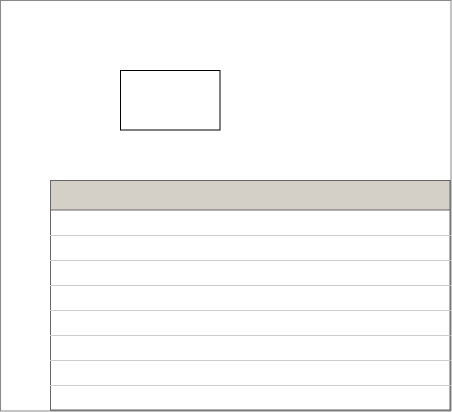
VISUALIZATION test  // 452x412
    Rectangle (120,70 100x60), colour toggle: MAIN.Q
    Table (50,180 400x230), data array: MAIN.arrWaarde
        p2232123230: MAIN.arrWaarde[1, INDEX]
        p511219082: MAIN.arrWaarde[2, INDEX]
END_VISUALIZATION

(* stored: Version 1.1.0.1, ProductVersion 3.1.4022.9
   Visu test: Id {ab0b0ec9-356e-4e4b-b5a3-1bed8871f2ba} *)
